PROGRAM UC_Measurements
VAR
	Puls: BOOL;
	Value: DINT:= 100; 
	Adjustment: DINT:= 10000; 
	FlowMeter: Measurement;
END_VAR

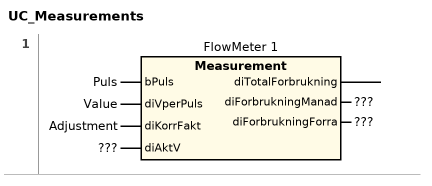
// NETWORK 1
FlowMeter 1(bPuls := Puls, diVperPuls := Value, diKorrFakt := Adjustment); // Measurement

END_PROGRAM

(* stored: Version 1.1.0.1, ProductVersion 3.1.4020.12
   POU UC_Measurements: Id {29be6c58-d715-4395-9896-8659d98e0df5}, SpecialFunc None *)
